(* IEC 61131-3 sources: Building-Automation/Car_Parking_Vending_System/plc, 6 files *)

(* ---- global_vars.st ---- *)
// Global Variables for Car Parking Vending System
// Version: 2.1.0
// Compatible with: Siemens S7-1200/1500, TIA Portal V17+

// =============================================================================
// SYSTEM ENUMERATIONS
// =============================================================================

TYPE SystemState :
(
    INIT := 0,              // System initialization
    IDLE := 1,              // Ready for operation
    PAYMENT := 2,           // Processing payment
    ENTRY := 3,             // Vehicle entry sequence
    PARKING := 4,           // Automated parking
    PARKED := 5,            // Vehicle stored
    RETRIEVAL := 6,         // Vehicle retrieval
    EXIT_SEQUENCE := 7,     // Vehicle exit
    MAINTENANCE := 8,       // Maintenance mode
    EMERGENCY := 9          // Emergency stop
);
END_TYPE;

TYPE ElevatorState :
(
    IDLE := 0,              // Elevator at rest
    MOVING_UP := 1,         // Moving upward
    MOVING_DOWN := 2,       // Moving downward
    POSITIONING := 3,       // Fine positioning
    LOADING := 4,           // Loading vehicle
    UNLOADING := 5,         // Unloading vehicle
    ERROR := 6              // Error state
);
END_TYPE;

TYPE PlatformState :
(
    HOME := 0,              // Home position
    MOVING_X := 1,          // Moving X axis
    MOVING_Y := 2,          // Moving Y axis
    POSITIONING := 3,       // Final positioning
    PICKING_UP := 4,        // Picking up vehicle
    DROPPING_OFF := 5,      // Dropping off vehicle
    ERROR := 6              // Error state
);
END_TYPE;

TYPE PaymentMethod :
(
    NONE := 0,              // No payment
    CASH := 1,              // Cash payment
    CREDIT_CARD := 2,       // Credit/Debit card
    RFID_CARD := 3,         // RFID membership card
    MOBILE_APP := 4,        // Mobile application
    QR_CODE := 5            // QR code payment
);
END_TYPE;

TYPE VehicleSize :
(
    COMPACT := 1,           // Small cars
    STANDARD := 2,          // Standard size
    SUV := 3,               // SUV/Large cars
    MOTORCYCLE := 4         // Motorcycles
);
END_TYPE;

// =============================================================================
// DIGITAL INPUTS (24V DC)
// =============================================================================

VAR_GLOBAL
    // Emergency stops and safety
    I_EmergencyStop_Main        AT %I0.0 : BOOL;   // Main emergency stop
    I_EmergencyStop_Level1      AT %I0.1 : BOOL;   // Level 1 emergency stop
    I_EmergencyStop_Level2      AT %I0.2 : BOOL;   // Level 2 emergency stop
    I_FireDetection_Zone1       AT %I0.3 : BOOL;   // Fire detector zone 1
    I_FireDetection_Zone2       AT %I0.4 : BOOL;   // Fire detector zone 2
    I_FireDetection_Zone3       AT %I0.5 : BOOL;   // Fire detector zone 3

    // Barrier positions
    I_EntryBarrier_OpenLimit    AT %I0.6 : BOOL;   // Entry barrier open
    I_EntryBarrier_CloseLimit   AT %I0.7 : BOOL;   // Entry barrier closed
    I_ExitBarrier_OpenLimit     AT %I1.0 : BOOL;   // Exit barrier open
    I_ExitBarrier_CloseLimit    AT %I1.1 : BOOL;   // Exit barrier closed

    // Vehicle detection
    I_VehiclePresent_Entry      AT %I1.2 : BOOL;   // Vehicle at entry
    I_VehiclePresent_Exit       AT %I1.3 : BOOL;   // Vehicle at exit
    I_VehiclePresent_Platform   AT %I1.4 : BOOL;   // Vehicle on platform
    I_VehiclePresent_Queue      AT %I1.5 : BOOL;   // Vehicle in queue

    // System positions
    I_Elevator1_Home            AT %I1.6 : BOOL;   // Elevator 1 home
    I_Elevator2_Home            AT %I1.7 : BOOL;   // Elevator 2 home
    I_Elevator3_Home            AT %I2.0 : BOOL;   // Elevator 3 home
    I_Platform_Home             AT %I2.1 : BOOL;   // Platform home position

    // System status
    I_DoorInterlocks_AllClosed  AT %I2.2 : BOOL;   // All doors closed
    I_HydraulicSystem_PressureOK AT %I2.3 : BOOL;  // Hydraulic pressure OK
    I_UPS_BatteryOK            AT %I2.4 : BOOL;   // UPS battery status
    I_Ventilation_StatusOK     AT %I2.5 : BOOL;   // Ventilation system OK
    I_MainPower_OK             AT %I2.6 : BOOL;   // Main power status
    I_NetworkConnection_OK     AT %I2.7 : BOOL;   // Network connectivity

    // Payment system inputs
    I_PaymentKiosk_Ready       AT %I3.0 : BOOL;   // Payment kiosk ready
    I_CashInserted             AT %I3.1 : BOOL;   // Cash payment received
    I_CardInserted             AT %I3.2 : BOOL;   // Card inserted
    I_RFIDCardPresent          AT %I3.3 : BOOL;   // RFID card detected
    I_QRCodeScanned            AT %I3.4 : BOOL;   // QR code scanned
    I_TicketPrinter_Ready      AT %I3.5 : BOOL;   // Ticket printer ready
    I_TicketPrinter_PaperOK    AT %I3.6 : BOOL;   // Printer paper OK
    I_ReceiptPrinter_Ready     AT %I3.7 : BOOL;   // Receipt printer ready

END_VAR;

// =============================================================================
// ANALOG INPUTS (4-20mA / 0-10V)
// =============================================================================

VAR_GLOBAL
    // Position feedback
    AI_Elevator1_Position       AT %IW0 : INT;     // Elevator 1 position (mm)
    AI_Elevator2_Position       AT %IW2 : INT;     // Elevator 2 position (mm)
    AI_Elevator3_Position       AT %IW4 : INT;     // Elevator 3 position (mm)
    AI_Platform_XPosition       AT %IW6 : INT;     // Platform X position (mm)
    AI_Platform_YPosition       AT %IW8 : INT;     // Platform Y position (mm)
    AI_Platform_ZPosition       AT %IW10 : INT;    // Platform Z position (mm)

    // System monitoring
    AI_HydraulicPressure        AT %IW12 : INT;    // Hydraulic pressure (bar)
    AI_Temperature_ControlRoom  AT %IW14 : INT;    // Control room temp (°C)
    AI_Humidity_ControlRoom     AT %IW16 : INT;    // Control room humidity (%)
    AI_LoadCell_PlatformWeight  AT %IW18 : INT;    // Platform load (kg)
    AI_PowerConsumption         AT %IW20 : INT;    // Power consumption (kW)
    AI_VibrationLevel          AT %IW22 : INT;    // Vibration level

    // Vehicle dimensions (from laser scanners)
    AI_VehicleLength           AT %IW24 : INT;    // Vehicle length (mm)
    AI_VehicleWidth            AT %IW26 : INT;    // Vehicle width (mm)
    AI_VehicleHeight           AT %IW28 : INT;    // Vehicle height (mm)
    AI_VehicleWeight           AT %IW30 : INT;    // Vehicle weight (kg)

END_VAR;

// =============================================================================
// DIGITAL OUTPUTS (24V DC)
// =============================================================================

VAR_GLOBAL
    // Barrier controls
    Q_EntryBarrier_Open         AT %Q0.0 : BOOL;   // Open entry barrier
    Q_EntryBarrier_Close        AT %Q0.1 : BOOL;   // Close entry barrier
    Q_ExitBarrier_Open          AT %Q0.2 : BOOL;   // Open exit barrier
    Q_ExitBarrier_Close         AT %Q0.3 : BOOL;   // Close exit barrier

    // Elevator controls
    Q_Elevator1_Enable          AT %Q0.4 : BOOL;   // Elevator 1 motor enable
    Q_Elevator2_Enable          AT %Q0.5 : BOOL;   // Elevator 2 motor enable
    Q_Elevator3_Enable          AT %Q0.6 : BOOL;   // Elevator 3 motor enable
    Q_Elevator1_Direction       AT %Q0.7 : BOOL;   // Elevator 1 direction
    Q_Elevator2_Direction       AT %Q1.0 : BOOL;   // Elevator 2 direction
    Q_Elevator3_Direction       AT %Q1.1 : BOOL;   // Elevator 3 direction

    // Platform controls
    Q_Platform_XEnable          AT %Q1.2 : BOOL;   // Platform X axis enable
    Q_Platform_YEnable          AT %Q1.3 : BOOL;   // Platform Y axis enable
    Q_Platform_ZEnable          AT %Q1.4 : BOOL;   // Platform Z axis enable
    Q_Platform_XDirection       AT %Q1.5 : BOOL;   // Platform X direction
    Q_Platform_YDirection       AT %Q1.6 : BOOL;   // Platform Y direction
    Q_Platform_ZDirection       AT %Q1.7 : BOOL;   // Platform Z direction

    // System controls
    Q_HydraulicPump            AT %Q2.0 : BOOL;   // Hydraulic pump start
    Q_VentilationFan           AT %Q2.1 : BOOL;   // Ventilation fan start
    Q_EmergencyLighting        AT %Q2.2 : BOOL;   // Emergency lighting
    Q_MainLighting             AT %Q2.3 : BOOL;   // Main lighting

    // Status indicators
    Q_StatusLight_Green        AT %Q2.4 : BOOL;   // Green status light
    Q_StatusLight_Yellow       AT %Q2.5 : BOOL;   // Yellow status light
    Q_StatusLight_Red          AT %Q2.6 : BOOL;   // Red status light
    Q_AlarmHorn               AT %Q2.7 : BOOL;   // Alarm horn

    // Door locks and safety
    Q_DoorLock_Entry          AT %Q3.0 : BOOL;   // Entry door lock
    Q_DoorLock_Exit           AT %Q3.1 : BOOL;   // Exit door lock
    Q_SafetyReset             AT %Q3.2 : BOOL;   // Safety system reset

    // Payment and printing
    Q_TicketPrinter_Print     AT %Q3.3 : BOOL;   // Print parking ticket
    Q_ReceiptPrinter_Print    AT %Q3.4 : BOOL;   // Print payment receipt
    Q_CashDispenser_Enable    AT %Q3.5 : BOOL;   // Cash change dispenser
    Q_CardReader_Enable       AT %Q3.6 : BOOL;   // Card reader enable
    Q_Display_Enable          AT %Q3.7 : BOOL;   // Customer display enable

    // System status outputs
    Q_SystemReady             AT %Q4.0 : BOOL;   // System ready indicator
    Q_SystemEnabled           AT %Q4.1 : BOOL;   // System enabled
    Q_MaintenanceMode         AT %Q4.2 : BOOL;   // Maintenance mode active
    Q_EmergencyActive         AT %Q4.3 : BOOL;   // Emergency mode active

END_VAR;

// =============================================================================
// ANALOG OUTPUTS (4-20mA / 0-10V)
// =============================================================================

VAR_GLOBAL
    // Speed references
    AQ_Elevator1_SpeedRef       AT %QW0 : INT;     // Elevator 1 speed ref
    AQ_Elevator2_SpeedRef       AT %QW2 : INT;     // Elevator 2 speed ref
    AQ_Elevator3_SpeedRef       AT %QW4 : INT;     // Elevator 3 speed ref
    AQ_Platform_XSpeedRef       AT %QW6 : INT;     // Platform X speed ref
    AQ_Platform_YSpeedRef       AT %QW8 : INT;     // Platform Y speed ref
    AQ_Platform_ZSpeedRef       AT %QW10 : INT;    // Platform Z speed ref

    // System controls
    AQ_HydraulicPressureRef     AT %QW12 : INT;    // Hydraulic pressure ref
    AQ_VentilationSpeedRef      AT %QW14 : INT;    // Ventilation speed ref
    AQ_LightingLevel           AT %QW16 : INT;    // Lighting level control

END_VAR;

// =============================================================================
// DATA STRUCTURES
// =============================================================================

TYPE ParkingSpace :
STRUCT
    Level : INT;                // Parking level (1-15)
    Position : INT;             // Position on level (1-20)
    Occupied : BOOL;            // Space occupied flag
    VehicleID : STRING[20];     // Vehicle identification
    ParkingTime : DATE_AND_TIME; // Time when parked
    VehicleType : VehicleSize;   // Vehicle size category
    ReservedFor : STRING[50];    // Reserved for specific customer
    MaintenanceRequired : BOOL;  // Maintenance flag
END_STRUCT;
END_TYPE;

TYPE Transaction :
STRUCT
    TransactionID : DINT;       // Unique transaction ID
    Timestamp : DATE_AND_TIME;  // Transaction timestamp
    CustomerID : STRING[50];    // Customer identification
    VehicleID : STRING[20];     // Vehicle license plate
    PaymentMethod : PaymentMethod; // Payment type used
    Amount : REAL;              // Payment amount
    ParkingDuration : TIME;     // Requested parking duration
    SpaceAssigned : ParkingSpace; // Assigned parking space
    Status : STRING[20];        // Transaction status
END_STRUCT;
END_TYPE;

TYPE SystemStatistics :
STRUCT
    TotalVehiclesParked : DINT;     // Total vehicles parked
    TotalVehiclesRetrieved : DINT;  // Total vehicles retrieved
    TotalRevenue : REAL;            // Total revenue generated
    AverageParkingTime : TIME;      // Average parking operation time
    AverageRetrievalTime : TIME;    // Average retrieval operation time
    SystemUptime : TIME;            // Total system uptime
    MaintenanceHours : TIME;        // Total maintenance time
    EmergencyStops : INT;           // Number of emergency stops
    PowerFailures : INT;            // Number of power failures
    LastMaintenanceDate : DATE;     // Last maintenance date
END_STRUCT;
END_TYPE;

TYPE ElevatorData :
STRUCT
    CurrentLevel : INT;         // Current elevator level
    TargetLevel : INT;          // Target level
    CurrentPosition : REAL;     // Current position (mm)
    TargetPosition : REAL;      // Target position (mm)
    Speed : REAL;               // Current speed (mm/s)
    State : ElevatorState;      // Current state
    LoadWeight : REAL;          // Current load weight (kg)
    LastService : DATE;         // Last service date
    OperationHours : TIME;      // Total operation hours
    FaultCode : INT;            // Current fault code
    Available : BOOL;           // Elevator available
END_STRUCT;
END_TYPE;

TYPE PlatformData :
STRUCT
    XPosition : REAL;           // Current X position (mm)
    YPosition : REAL;           // Current Y position (mm)
    ZPosition : REAL;           // Current Z position (mm)
    XTarget : REAL;             // Target X position
    YTarget : REAL;             // Target Y position
    ZTarget : REAL;             // Target Z position
    State : PlatformState;      // Current platform state
    LoadWeight : REAL;          // Current load weight (kg)
    VehicleSecured : BOOL;      // Vehicle properly secured
    LastCalibration : DATE_AND_TIME; // Last calibration
    FaultCode : INT;            // Current fault code
    Available : BOOL;           // Platform available
END_STRUCT;
END_TYPE;

// =============================================================================
// GLOBAL SYSTEM VARIABLES
// =============================================================================

VAR_GLOBAL
    // Parking space array (15 levels × 20 spaces = 300 total)
    ParkingSpaces : ARRAY[1..15, 1..20] OF ParkingSpace;

    // System statistics and monitoring
    SystemStats : SystemStatistics;

    // Equipment data
    Elevator1 : ElevatorData;
    Elevator2 : ElevatorData;
    Elevator3 : ElevatorData;
    Platform : PlatformData;

    // Current transaction
    CurrentTransaction : Transaction;
    TransactionCounter : DINT := 0;

    // System configuration
    MaxVehicleLength : REAL := 5200.0;     // mm
    MaxVehicleWidth : REAL := 2100.0;      // mm
    MaxVehicleHeight : REAL := 1800.0;     // mm
    MaxVehicleWeight : REAL := 3500.0;     // kg

    // Pricing structure
    HourlyRate : REAL := 2.50;             // Currency per hour
    DailyRate : REAL := 15.00;             // Currency per day
    MonthlyRate : REAL := 150.00;          // Currency per month

    // Operating parameters
    ElevatorSpeed : REAL := 2500.0;        // mm/s
    PlatformSpeed : REAL := 1500.0;        // mm/s
    PositioningTolerance : REAL := 5.0;    // mm

    // System timers and counters
    SystemStartTime : DATE_AND_TIME;
    LastTransactionTime : DATE_AND_TIME;
    NextMaintenanceTime : DATE_AND_TIME;

    // Queue management
    WaitingVehicles : INT := 0;
    MaxQueueLength : INT := 10;
    EstimatedWaitTime : TIME;

    // Performance monitoring
    SystemEfficiency : REAL;               // 0-100%
    EnergyConsumption : REAL;              // kWh
    ThroughputPerHour : REAL;              // vehicles/hour

    // Alarm and event logging
    AlarmBuffer : ARRAY[1..100] OF STRING[200];
    EventBuffer : ARRAY[1..1000] OF STRING[200];
    AlarmIndex : INT := 0;
    EventIndex : INT := 0;

    // Communication and networking
    HMI_Connected : BOOL := FALSE;
    Database_Connected : BOOL := FALSE;
    PaymentGateway_Connected : BOOL := FALSE;
    RemoteMonitoring_Connected : BOOL := FALSE;

    // Weather and environmental
    OutdoorTemperature : REAL;
    WindSpeed : REAL;
    RainIntensity : REAL;

END_VAR;

// =============================================================================
// SYSTEM CONSTANTS
// =============================================================================

VAR_GLOBAL CONSTANT
    SYSTEM_VERSION : STRING := '2.1.0';
    MAX_PARKING_LEVELS : INT := 15;
    SPACES_PER_LEVEL : INT := 20;
    TOTAL_PARKING_SPACES : INT := 300;

    // Safety limits
    MAX_ELEVATOR_SPEED : REAL := 3000.0;   // mm/s
    MAX_PLATFORM_SPEED : REAL := 2000.0;   // mm/s
    EMERGENCY_STOP_TIME : TIME := T#2s;

    // Operational timeouts
    PAYMENT_TIMEOUT : TIME := T#120s;
    ENTRY_TIMEOUT : TIME := T#60s;
    PARKING_TIMEOUT : TIME := T#300s;
    RETRIEVAL_TIMEOUT : TIME := T#300s;
    EXIT_TIMEOUT : TIME := T#90s;

    // Communication timeouts
    HMI_TIMEOUT : TIME := T#10s;
    DATABASE_TIMEOUT : TIME := T#30s;
    NETWORK_TIMEOUT : TIME := T#15s;

END_VAR;

(* ---- elevator_controller.st ---- *)
FUNCTION_BLOCK ElevatorController
VAR_INPUT
    ElevatorNumber : INT;               // Elevator number (1, 2, or 3)
    TargetLevel : INT;                  // Target level (1-15)
    Execute : BOOL;                     // Execute movement command
    Stop : BOOL;                        // Emergency stop
    Reset : BOOL;                       // Reset elevator
    ManualMode : BOOL;                  // Manual operation mode
    ManualDirection : BOOL;             // Manual direction (TRUE=up, FALSE=down)
    ManualSpeed : REAL;                 // Manual speed reference
END_VAR

VAR_OUTPUT
    Done : BOOL;                        // Movement completed
    Busy : BOOL;                        // Movement in progress
    Error : BOOL;                       // Error condition
    ErrorID : INT;                      // Error identification code
    CurrentLevel : INT;                 // Current elevator level
    CurrentPosition : REAL;             // Current position (mm)
    AtLevel : BOOL;                     // At target level
    DoorOpen : BOOL;                    // Door open status
    Available : BOOL;                   // Elevator available for use
    LoadWeight : REAL;                  // Current load weight
    MotorSpeed : REAL;                  // Current motor speed
END_VAR

VAR
    // Control state machine
    state : INT := 0;
    previousState : INT;
    stateTimer : TON;
    movementTimer : TON;

    // Position and motion control
    currentPos : REAL;                  // Current position in mm
    targetPos : REAL;                   // Target position in mm
    homePosition : REAL := 0.0;         // Ground level position
    levelHeight : REAL := 3000.0;       // Height per level (mm)
    positionTolerance : REAL := 20.0;   // Position tolerance (mm)

    // Motion parameters
    maxSpeed : REAL := 2500.0;          // Maximum speed (mm/s)
    acceleration : REAL := 500.0;       // Acceleration (mm/s²)
    deceleration : REAL := 750.0;       // Deceleration (mm/s²)
    currentSpeed : REAL := 0.0;         // Current speed
    targetSpeed : REAL := 0.0;          // Target speed

    // Safety and monitoring
    safetyOK : BOOL := TRUE;
    overloadDetected : BOOL := FALSE;
    doorInterlockOK : BOOL := TRUE;
    emergencyStopActive : BOOL := FALSE;

    // Door control
    doorState : INT := 0;               // 0=closed, 1=opening, 2=open, 3=closing
    doorTimer : TON;
    doorTimeout : TIME := T#10s;

    // Maintenance and diagnostics
    totalOperationTime : TIME;
    totalDistance : REAL := 0.0;
    cycleCount : DINT := 0;
    lastMaintenanceDistance : REAL := 0.0;
    maintenanceRequired : BOOL := FALSE;

    // Error handling
    errorHistory : ARRAY[1..10] OF INT;
    errorIndex : INT := 1;
    retryCount : INT := 0;
    maxRetries : INT := 3;

    // Performance monitoring
    averageSpeed : REAL;
    lastMovementTime : TIME;
    efficiency : REAL := 100.0;

END_VAR

// Input validation
IF ElevatorNumber < 1 OR ElevatorNumber > 3 THEN
    Error := TRUE;
    ErrorID := 5001; // Invalid elevator number
    Available := FALSE;
    RETURN;
END_IF;

IF TargetLevel < 1 OR TargetLevel > MAX_PARKING_LEVELS THEN
    Error := TRUE;
    ErrorID := 5002; // Invalid target level
    RETURN;
END_IF;

// Get current position based on elevator number
CASE ElevatorNumber OF
    1: currentPos := SCALE_INT_TO_REAL(AI_Elevator1_Position, 0.0, 45000.0);
    2: currentPos := SCALE_INT_TO_REAL(AI_Elevator2_Position, 0.0, 45000.0);
    3: currentPos := SCALE_INT_TO_REAL(AI_Elevator3_Position, 0.0, 45000.0);
END_CASE;

CurrentPosition := currentPos;
LoadWeight := SCALE_INT_TO_REAL(AI_LoadCell_PlatformWeight, 0.0, 5000.0);

// Calculate current level
CurrentLevel := REAL_TO_INT((currentPos / levelHeight) + 1);
IF CurrentLevel < 1 THEN CurrentLevel := 1; END_IF;
IF CurrentLevel > MAX_PARKING_LEVELS THEN CurrentLevel := MAX_PARKING_LEVELS; END_IF;

// Safety checks
safetyOK := NOT I_EmergencyStop_Main AND
            NOT I_EmergencyStop_Level1 AND
            NOT I_EmergencyStop_Level2 AND
            I_HydraulicSystem_PressureOK AND
            I_UPS_BatteryOK;

overloadDetected := LoadWeight > 4000.0; // 4000kg limit
doorInterlockOK := I_DoorInterlocks_AllClosed;
emergencyStopActive := Stop OR NOT safetyOK;

// Emergency stop handling
IF emergencyStopActive THEN
    state := 90; // Emergency stop state
    targetSpeed := 0.0;
    Error := TRUE;
    ErrorID := 5010;
END_IF;

// Reset handling
IF Reset AND state = 90 THEN
    state := 0; // Reset to idle
    Error := FALSE;
    ErrorID := 0;
    retryCount := 0;
END_IF;

// Calculate target position
targetPos := (TargetLevel - 1) * levelHeight;

// Check if at target level
AtLevel := ABS(currentPos - targetPos) <= positionTolerance;

// Execute movement command
IF Execute AND NOT Busy AND state = 0 AND safetyOK THEN
    IF NOT AtLevel THEN
        Busy := TRUE;
        Done := FALSE;
        state := 10; // Start movement
        movementTimer(IN := TRUE, PT := T#0s);
        cycleCount := cycleCount + 1;
    ELSE
        Done := TRUE; // Already at target
    END_IF;
END_IF;

// Manual mode handling
IF ManualMode AND state = 0 AND safetyOK THEN
    state := 80; // Manual mode
    Busy := TRUE;
END_IF;

// Main state machine
CASE state OF

    0: // IDLE
        Busy := FALSE;
        Available := TRUE AND safetyOK AND NOT maintenanceRequired;
        targetSpeed := 0.0;

        // Check for maintenance requirements
        IF (totalDistance - lastMaintenanceDistance) > 100000000.0 THEN // 100km
            maintenanceRequired := TRUE;
            Available := FALSE;
        END_IF;

    // =============================================================================
    // MOVEMENT SEQUENCE (States 10-49)
    // =============================================================================

    10: // PREPARE_FOR_MOVEMENT
        Available := FALSE;

        // Ensure doors are closed
        IF NOT doorInterlockOK THEN
            state := 11; // Close doors first
        ELSE
            state := 12; // Doors already closed
        END_IF;

    11: // CLOSE_DOORS
        doorState := 3; // Closing
        doorTimer(IN := TRUE, PT := doorTimeout);

        IF doorInterlockOK THEN
            doorState := 0; // Closed
            state := 12;
            doorTimer(IN := FALSE);
        ELSIF doorTimer.Q THEN
            Error := TRUE;
            ErrorID := 5011; // Door close timeout
            state := 91;
            doorTimer(IN := FALSE);
        END_IF;

    12: // START_MOVEMENT
        // Enable motor based on elevator number
        CASE ElevatorNumber OF
            1: Q_Elevator1_Enable := TRUE;
            2: Q_Elevator2_Enable := TRUE;
            3: Q_Elevator3_Enable := TRUE;
        END_CASE;

        // Determine direction
        IF targetPos > currentPos THEN
            // Moving up
            CASE ElevatorNumber OF
                1: Q_Elevator1_Direction := TRUE;
                2: Q_Elevator2_Direction := TRUE;
                3: Q_Elevator3_Direction := TRUE;
            END_CASE;
        ELSE
            // Moving down
            CASE ElevatorNumber OF
                1: Q_Elevator1_Direction := FALSE;
                2: Q_Elevator2_Direction := FALSE;
                3: Q_Elevator3_Direction := FALSE;
            END_CASE;
        END_IF;

        state := 13; // Accelerate

    13: // ACCELERATE
        // Calculate required speed
        IF ABS(targetPos - currentPos) > 1000.0 THEN
            targetSpeed := maxSpeed; // Full speed for long distances
        ELSE
            targetSpeed := maxSpeed * 0.5; // Half speed for short distances
        END_IF;

        // Accelerate to target speed
        IF currentSpeed < targetSpeed THEN
            currentSpeed := currentSpeed + (acceleration * 0.1); // 100ms cycle
            IF currentSpeed > targetSpeed THEN
                currentSpeed := targetSpeed;
            END_IF;
        END_IF;

        // Check if close to target for deceleration
        IF ABS(targetPos - currentPos) <= (currentSpeed * currentSpeed) / (2.0 * deceleration) THEN
            state := 14; // Start deceleration
        END_IF;

        // Safety check during movement
        IF NOT safetyOK OR overloadDetected THEN
            state := 90; // Emergency stop
        END_IF;

    14: // DECELERATE
        // Calculate deceleration distance
        targetSpeed := SQRT(2.0 * deceleration * ABS(targetPos - currentPos));

        IF targetSpeed < 100.0 THEN
            targetSpeed := 100.0; // Minimum speed for positioning
        END_IF;

        // Decelerate
        IF currentSpeed > targetSpeed THEN
            currentSpeed := currentSpeed - (deceleration * 0.1);
            IF currentSpeed < targetSpeed THEN
                currentSpeed := targetSpeed;
            END_IF;
        END_IF;

        // Check if at target position
        IF ABS(targetPos - currentPos) <= positionTolerance THEN
            state := 15; // Stop
        END_IF;

        // Timeout check
        IF movementTimer.ET > T#300s THEN
            Error := TRUE;
            ErrorID := 5012; // Movement timeout
            state := 91;
        END_IF;

    15: // STOP_AT_TARGET
        targetSpeed := 0.0;
        currentSpeed := 0.0;

        // Stop motor
        CASE ElevatorNumber OF
            1: Q_Elevator1_Enable := FALSE;
            2: Q_Elevator2_Enable := FALSE;
            3: Q_Elevator3_Enable := FALSE;
        END_CASE;

        stateTimer(IN := TRUE, PT := T#2s);

        IF stateTimer.Q THEN
            state := 16; // Final positioning
            stateTimer(IN := FALSE);
        END_IF;

    16: // FINE_POSITIONING
        // Fine positioning at very low speed
        IF ABS(targetPos - currentPos) > 5.0 THEN
            CASE ElevatorNumber OF
                1: Q_Elevator1_Enable := TRUE;
                2: Q_Elevator2_Enable := TRUE;
                3: Q_Elevator3_Enable := TRUE;
            END_CASE;

            currentSpeed := 50.0; // Very slow speed
            targetSpeed := 50.0;
        ELSE
            state := 17; // Positioning complete
        END_IF;

        stateTimer(IN := TRUE, PT := T#30s);
        IF stateTimer.Q THEN
            state := 17; // Timeout - accept current position
            stateTimer(IN := FALSE);
        END_IF;

    17: // POSITIONING_COMPLETE
        // Final stop
        targetSpeed := 0.0;
        currentSpeed := 0.0;

        CASE ElevatorNumber OF
            1: Q_Elevator1_Enable := FALSE;
            2: Q_Elevator2_Enable := FALSE;
            3: Q_Elevator3_Enable := FALSE;
        END_CASE;

        // Update statistics
        lastMovementTime := movementTimer.ET;
        totalDistance := totalDistance + ABS(targetPos - currentPos);
        averageSpeed := ABS(targetPos - currentPos) / TIME_TO_REAL(lastMovementTime);

        state := 20; // Open doors

    20: // OPEN_DOORS
        doorState := 1; // Opening
        doorTimer(IN := TRUE, PT := doorTimeout);

        stateTimer(IN := TRUE, PT := T#2s);

        IF stateTimer.Q THEN
            doorState := 2; // Open
            DoorOpen := TRUE;
            state := 30; // Movement complete
            doorTimer(IN := FALSE);
            stateTimer(IN := FALSE);
        ELSIF doorTimer.Q THEN
            // Door open timeout - continue anyway
            DoorOpen := FALSE;
            state := 30;
            doorTimer(IN := FALSE);
        END_IF;

    30: // MOVEMENT_COMPLETE
        Done := TRUE;
        Busy := FALSE;
        Available := TRUE;
        AtLevel := TRUE;

        // Log successful movement
        LogEvent('ELEVATOR_MOVEMENT', 'Elevator ' + INT_TO_STRING(ElevatorNumber) +
                 ' moved to level ' + INT_TO_STRING(TargetLevel) +
                 ' in ' + TIME_TO_STRING(lastMovementTime));

        state := 0; // Return to idle

    // =============================================================================
    // MANUAL MODE (States 80-89)
    // =============================================================================

    80: // MANUAL_OPERATION
        Available := FALSE;

        IF NOT ManualMode THEN
            state := 0; // Exit manual mode
            targetSpeed := 0.0;
        ELSE
            // Enable motor
            CASE ElevatorNumber OF
                1: Q_Elevator1_Enable := TRUE;
                   Q_Elevator1_Direction := ManualDirection;
                2: Q_Elevator2_Enable := TRUE;
                   Q_Elevator2_Direction := ManualDirection;
                3: Q_Elevator3_Enable := TRUE;
                   Q_Elevator3_Direction := ManualDirection;
            END_CASE;

            targetSpeed := ManualSpeed;
            currentSpeed := ManualSpeed;

            // Safety limits in manual mode
            IF currentPos <= 0.0 AND NOT ManualDirection THEN
                targetSpeed := 0.0; // At bottom limit
            ELSIF currentPos >= 45000.0 AND ManualDirection THEN
                targetSpeed := 0.0; // At top limit
            END_IF;
        END_IF;

    // =============================================================================
    // ERROR STATES (States 90-99)
    // =============================================================================

    90: // EMERGENCY_STOP
        targetSpeed := 0.0;
        currentSpeed := 0.0;
        Available := FALSE;
        Error := TRUE;

        // Stop motor immediately
        CASE ElevatorNumber OF
            1: Q_Elevator1_Enable := FALSE;
            2: Q_Elevator2_Enable := FALSE;
            3: Q_Elevator3_Enable := FALSE;
        END_CASE;

        // Log emergency stop
        LogError(ErrorID, 'Emergency stop - Elevator ' + INT_TO_STRING(ElevatorNumber));

        // Stay in this state until reset

    91: // ERROR_WITH_RETRY
        Error := TRUE;
        Available := FALSE;
        targetSpeed := 0.0;

        // Stop motor
        CASE ElevatorNumber OF
            1: Q_Elevator1_Enable := FALSE;
            2: Q_Elevator2_Enable := FALSE;
            3: Q_Elevator3_Enable := FALSE;
        END_CASE;

        // Record error
        errorHistory[errorIndex] := ErrorID;
        errorIndex := errorIndex + 1;
        IF errorIndex > 10 THEN errorIndex := 1; END_IF;

        // Retry logic
        IF retryCount < maxRetries AND safetyOK THEN
            retryCount := retryCount + 1;
            stateTimer(IN := TRUE, PT := T#10s);

            IF stateTimer.Q THEN
                state := 10; // Retry movement
                Error := FALSE;
                ErrorID := 0;
                stateTimer(IN := FALSE);
            END_IF;
        ELSE
            state := 90; // Give up, require manual reset
        END_IF;

END_CASE;

// Set speed reference outputs
CASE ElevatorNumber OF
    1: AQ_Elevator1_SpeedRef := REAL_TO_INT(currentSpeed);
    2: AQ_Elevator2_SpeedRef := REAL_TO_INT(currentSpeed);
    3: AQ_Elevator3_SpeedRef := REAL_TO_INT(currentSpeed);
END_CASE;

// Update motor speed output for monitoring
MotorSpeed := currentSpeed;

// Update total operation time
totalOperationTime := totalOperationTime + T#100ms;

// Update elevator data structure
CASE ElevatorNumber OF
    1: Elevator1.CurrentLevel := CurrentLevel;
       Elevator1.CurrentPosition := currentPos;
       Elevator1.TargetLevel := TargetLevel;
       Elevator1.TargetPosition := targetPos;
       Elevator1.Speed := currentSpeed;
       Elevator1.LoadWeight := LoadWeight;
       Elevator1.Available := Available;
       Elevator1.FaultCode := ErrorID;
       Elevator1.OperationHours := totalOperationTime;

    2: Elevator2.CurrentLevel := CurrentLevel;
       Elevator2.CurrentPosition := currentPos;
       Elevator2.TargetLevel := TargetLevel;
       Elevator2.TargetPosition := targetPos;
       Elevator2.Speed := currentSpeed;
       Elevator2.LoadWeight := LoadWeight;
       Elevator2.Available := Available;
       Elevator2.FaultCode := ErrorID;
       Elevator2.OperationHours := totalOperationTime;

    3: Elevator3.CurrentLevel := CurrentLevel;
       Elevator3.CurrentPosition := currentPos;
       Elevator3.TargetLevel := TargetLevel;
       Elevator3.TargetPosition := targetPos;
       Elevator3.Speed := currentSpeed;
       Elevator3.LoadWeight := LoadWeight;
       Elevator3.Available := Available;
       Elevator3.FaultCode := ErrorID;
       Elevator3.OperationHours := totalOperationTime;
END_CASE;

// Store previous state for debugging
previousState := state;

END_FUNCTION_BLOCK

(* ---- parking_controller.st ---- *)
FUNCTION_BLOCK ParkingController
VAR_INPUT
    Execute : BOOL;                     // Execute parking sequence
    VehicleRetrievalRequest : BOOL;     // Vehicle retrieval request
    CustomerID : STRING[50];            // Customer identification
    VehicleID : STRING[20];             // Vehicle license plate
    PaymentValidated : BOOL;            // Payment validation status
END_VAR

VAR_OUTPUT
    Done : BOOL;                        // Operation completed
    Busy : BOOL;                        // Operation in progress
    Error : BOOL;                       // Error occurred
    ErrorID : INT;                      // Error identification
    AssignedSpace : ParkingSpace;       // Assigned parking space
    EstimatedTime : TIME;               // Estimated completion time
END_VAR

VAR
    // State machine for parking operations
    state : INT := 0;
    stepTimer : TON;
    operationTimer : TON;

    // Vehicle handling
    vehicleDimensions : VehicleDimensions;
    optimalSpace : ParkingSpace;
    selectedElevator : INT;

    // Position control
    targetLevel : INT;
    targetXPosition : REAL;
    targetYPosition : REAL;
    currentOperation : STRING[50];

    // Safety and monitoring
    platformSecure : BOOL;
    elevatorReady : BOOL;
    spaceAvailable : BOOL;

    // Performance tracking
    operationStartTime : DATE_AND_TIME;
    parkingSequenceTime : TIME;
    retrievalSequenceTime : TIME;

    // Error handling
    retryCount : INT := 0;
    maxRetries : INT := 3;
    lastErrorTime : DATE_AND_TIME;

END_VAR

// Vehicle dimensions structure
TYPE VehicleDimensions :
STRUCT
    Length : REAL;
    Width : REAL;
    Height : REAL;
    Weight : REAL;
    VehicleType : VehicleSize;
END_STRUCT;
END_TYPE;

// Main execution logic
IF Execute AND NOT Busy THEN
    Busy := TRUE;
    Done := FALSE;
    Error := FALSE;
    state := 10; // Start parking sequence
    operationStartTime := GetSystemTime();
    operationTimer(IN := TRUE, PT := T#0s);
ELSIF VehicleRetrievalRequest AND NOT Busy THEN
    Busy := TRUE;
    Done := FALSE;
    Error := FALSE;
    state := 50; // Start retrieval sequence
    operationStartTime := GetSystemTime();
    operationTimer(IN := TRUE, PT := T#0s);
END_IF;

// Main state machine
CASE state OF

    0: // IDLE
        Busy := FALSE;
        Done := FALSE;
        Error := FALSE;
        currentOperation := 'IDLE';

    // =============================================================================
    // PARKING SEQUENCE (States 10-39)
    // =============================================================================

    10: // SCAN_VEHICLE_DIMENSIONS
        currentOperation := 'SCANNING_VEHICLE';

        // Get vehicle dimensions from laser scanners
        vehicleDimensions.Length := SCALE_INT_TO_REAL(AI_VehicleLength, 0.0, 6000.0);
        vehicleDimensions.Width := SCALE_INT_TO_REAL(AI_VehicleWidth, 0.0, 2500.0);
        vehicleDimensions.Height := SCALE_INT_TO_REAL(AI_VehicleHeight, 0.0, 2000.0);
        vehicleDimensions.Weight := SCALE_INT_TO_REAL(AI_VehicleWeight, 0.0, 5000.0);

        // Determine vehicle type
        IF vehicleDimensions.Length <= 4200.0 AND vehicleDimensions.Width <= 1800.0 THEN
            vehicleDimensions.VehicleType := COMPACT;
        ELSIF vehicleDimensions.Length <= 5200.0 AND vehicleDimensions.Width <= 2100.0 THEN
            vehicleDimensions.VehicleType := STANDARD;
        ELSIF vehicleDimensions.Height <= 1200.0 THEN
            vehicleDimensions.VehicleType := MOTORCYCLE;
        ELSE
            vehicleDimensions.VehicleType := SUV;
        END_IF;

        // Validate vehicle dimensions
        IF vehicleDimensions.Length > MaxVehicleLength OR
           vehicleDimensions.Width > MaxVehicleWidth OR
           vehicleDimensions.Height > MaxVehicleHeight OR
           vehicleDimensions.Weight > MaxVehicleWeight THEN
            Error := TRUE;
            ErrorID := 2001; // Vehicle too large
            state := 90; // Error handling
        ELSE
            state := 11; // Continue to space finding
        END_IF;

    11: // FIND_OPTIMAL_SPACE
        currentOperation := 'FINDING_PARKING_SPACE';

        IF FindOptimalParkingSpace() THEN
            state := 12; // Space found
        ELSE
            Error := TRUE;
            ErrorID := 2002; // No available space
            state := 90; // Error handling
        END_IF;

    12: // PREPARE_PLATFORM
        currentOperation := 'PREPARING_PLATFORM';

        // Ensure platform is at home position
        IF I_Platform_Home THEN
            Q_Platform_XEnable := TRUE;
            Q_Platform_YEnable := TRUE;
            Q_Platform_ZEnable := TRUE;
            state := 13;
        ELSE
            // Move platform to home position
            MovePlatformToHome();
        END_IF;

    13: // POSITION_VEHICLE_ON_PLATFORM
        currentOperation := 'POSITIONING_VEHICLE';

        stepTimer(IN := TRUE, PT := T#30s);

        // Check if vehicle is properly positioned
        IF I_VehiclePresent_Platform AND
           ABS(AI_Platform_XPosition - 3000) < 50 AND  // Center X position
           ABS(AI_Platform_YPosition - 7500) < 50 THEN // Center Y position
            platformSecure := TRUE;
            state := 14;
            stepTimer(IN := FALSE);
        ELSIF stepTimer.Q THEN
            Error := TRUE;
            ErrorID := 2003; // Vehicle positioning timeout
            state := 90;
            stepTimer(IN := FALSE);
        END_IF;

    14: // SECURE_VEHICLE
        currentOperation := 'SECURING_VEHICLE';

        // Activate platform securing mechanisms
        Q_Platform_ZEnable := TRUE;
        AQ_Platform_ZSpeedRef := 100; // Slow speed for securing

        stepTimer(IN := TRUE, PT := T#10s);

        // Check if vehicle is secured (weight on platform)
        IF AI_LoadCell_PlatformWeight > 500 THEN // Minimum 500kg
            Platform.VehicleSecured := TRUE;
            state := 15;
            stepTimer(IN := FALSE);
        ELSIF stepTimer.Q THEN
            Error := TRUE;
            ErrorID := 2004; // Vehicle securing failed
            state := 90;
            stepTimer(IN := FALSE);
        END_IF;

    15: // SELECT_ELEVATOR
        currentOperation := 'SELECTING_ELEVATOR';

        selectedElevator := SelectOptimalElevator();

        IF selectedElevator > 0 THEN
            state := 16;
        ELSE
            Error := TRUE;
            ErrorID := 2005; // No elevator available
            state := 90;
        END_IF;

    16: // MOVE_TO_ELEVATOR
        currentOperation := 'MOVING_TO_ELEVATOR';

        // Calculate elevator loading position
        CASE selectedElevator OF
            1: targetXPosition := 1500.0; // Elevator 1 position
            2: targetXPosition := 3000.0; // Elevator 2 position
            3: targetXPosition := 4500.0; // Elevator 3 position
        END_CASE;

        targetYPosition := 2000.0; // Elevator loading position

        MovePlatformToPosition(targetXPosition, targetYPosition, 0.0);

        // Check if platform reached elevator
        IF ABS(AI_Platform_XPosition - targetXPosition) < 20 AND
           ABS(AI_Platform_YPosition - targetYPosition) < 20 THEN
            state := 17;
        END_IF;

    17: // LOAD_INTO_ELEVATOR
        currentOperation := 'LOADING_INTO_ELEVATOR';

        stepTimer(IN := TRUE, PT := T#60s);

        // Enable selected elevator
        CASE selectedElevator OF
            1: Q_Elevator1_Enable := TRUE;
            2: Q_Elevator2_Enable := TRUE;
            3: Q_Elevator3_Enable := TRUE;
        END_CASE;

        // Transfer vehicle to elevator
        Q_Platform_YEnable := TRUE;
        Q_Platform_YDirection := TRUE; // Move forward into elevator
        AQ_Platform_YSpeedRef := 500; // Slow speed for precision

        // Check if loading complete
        IF ABS(AI_Platform_YPosition - 1000.0) < 10 THEN // Inside elevator
            state := 18;
            stepTimer(IN := FALSE);
        ELSIF stepTimer.Q THEN
            Error := TRUE;
            ErrorID := 2006; // Elevator loading timeout
            state := 90;
            stepTimer(IN := FALSE);
        END_IF;

    18: // MOVE_TO_PARKING_LEVEL
        currentOperation := 'MOVING_TO_LEVEL';

        targetLevel := optimalSpace.Level;

        MoveElevatorToLevel(selectedElevator, targetLevel);

        // Check if elevator reached target level
        CASE selectedElevator OF
            1: IF ABS(AI_Elevator1_Position - (targetLevel * 3000)) < 50 THEN
                   state := 19;
               END_IF;
            2: IF ABS(AI_Elevator2_Position - (targetLevel * 3000)) < 50 THEN
                   state := 19;
               END_IF;
            3: IF ABS(AI_Elevator3_Position - (targetLevel * 3000)) < 50 THEN
                   state := 19;
               END_IF;
        END_CASE;

    19: // UNLOAD_FROM_ELEVATOR
        currentOperation := 'UNLOADING_FROM_ELEVATOR';

        stepTimer(IN := TRUE, PT := T#60s);

        // Move platform out of elevator to parking level
        Q_Platform_YDirection := FALSE; // Move backward out of elevator
        AQ_Platform_YSpeedRef := 500; // Slow speed

        // Calculate target position on parking level
        targetXPosition := optimalSpace.Position * 300.0; // 300mm spacing
        targetYPosition := 7500.0; // Level corridor position

        IF ABS(AI_Platform_YPosition - targetYPosition) < 20 THEN
            state := 20;
            stepTimer(IN := FALSE);
        ELSIF stepTimer.Q THEN
            Error := TRUE;
            ErrorID := 2007; // Elevator unloading timeout
            state := 90;
            stepTimer(IN := FALSE);
        END_IF;

    20: // MOVE_TO_PARKING_SPACE
        currentOperation := 'MOVING_TO_SPACE';

        MovePlatformToPosition(targetXPosition, targetYPosition, 0.0);

        // Check if platform reached parking space
        IF ABS(AI_Platform_XPosition - targetXPosition) < 10 AND
           ABS(AI_Platform_YPosition - targetYPosition) < 10 THEN
            state := 21;
        END_IF;

    21: // DEPOSIT_VEHICLE
        currentOperation := 'DEPOSITING_VEHICLE';

        stepTimer(IN := TRUE, PT := T#30s);

        // Lower platform to deposit vehicle
        Q_Platform_ZDirection := FALSE; // Move down
        AQ_Platform_ZSpeedRef := 200; // Very slow for safety

        // Check if vehicle deposited (reduced weight on platform)
        IF AI_LoadCell_PlatformWeight < 100 THEN // Most weight removed
            state := 22;
            stepTimer(IN := FALSE);
        ELSIF stepTimer.Q THEN
            Error := TRUE;
            ErrorID := 2008; // Vehicle deposit timeout
            state := 90;
            stepTimer(IN := FALSE);
        END_IF;

    22: // UPDATE_PARKING_RECORD
        currentOperation := 'UPDATING_RECORDS';

        // Mark space as occupied
        ParkingSpaces[optimalSpace.Level, optimalSpace.Position].Occupied := TRUE;
        ParkingSpaces[optimalSpace.Level, optimalSpace.Position].VehicleID := VehicleID;
        ParkingSpaces[optimalSpace.Level, optimalSpace.Position].ParkingTime := GetSystemTime();
        ParkingSpaces[optimalSpace.Level, optimalSpace.Position].VehicleType := vehicleDimensions.VehicleType;

        // Update transaction record
        CurrentTransaction.SpaceAssigned := optimalSpace;
        CurrentTransaction.Status := 'PARKED';

        // Update system statistics
        SystemStats.TotalVehiclesParked := SystemStats.TotalVehiclesParked + 1;
        parkingSequenceTime := operationTimer.ET;

        // Calculate average parking time
        SystemStats.AverageParkingTime :=
            DINT_TO_TIME((TIME_TO_DINT(SystemStats.AverageParkingTime) *
                         (SystemStats.TotalVehiclesParked - 1) +
                         TIME_TO_DINT(parkingSequenceTime)) /
                         SystemStats.TotalVehiclesParked);

        state := 23; // Return platform home

    23: // RETURN_PLATFORM_HOME
        currentOperation := 'RETURNING_HOME';

        MovePlatformToHome();

        IF I_Platform_Home THEN
            state := 30; // Parking sequence complete
        END_IF;

    30: // PARKING_COMPLETE
        currentOperation := 'PARKING_COMPLETE';
        AssignedSpace := optimalSpace;
        Done := TRUE;
        Busy := FALSE;
        state := 0; // Return to idle

        // Log successful parking
        LogEvent('PARKING_SUCCESS', VehicleID + ' parked at Level ' +
                 INT_TO_STRING(optimalSpace.Level) + ' Position ' +
                 INT_TO_STRING(optimalSpace.Position));

    // =============================================================================
    // RETRIEVAL SEQUENCE (States 50-89)
    // =============================================================================

    50: // FIND_PARKED_VEHICLE
        currentOperation := 'FINDING_VEHICLE';

        IF FindParkedVehicle(VehicleID) THEN
            state := 51;
        ELSE
            Error := TRUE;
            ErrorID := 3001; // Vehicle not found
            state := 90;
        END_IF;

    51: // PREPARE_FOR_RETRIEVAL
        currentOperation := 'PREPARING_RETRIEVAL';

        // Select optimal elevator for retrieval
        selectedElevator := SelectOptimalElevator();

        // Ensure platform is at home
        IF I_Platform_Home THEN
            state := 52;
        ELSE
            MovePlatformToHome();
        END_IF;

    52: // MOVE_TO_RETRIEVAL_LEVEL
        currentOperation := 'MOVING_TO_LEVEL';

        targetLevel := optimalSpace.Level;
        MoveElevatorToLevel(selectedElevator, targetLevel);

        // Check if elevator reached target level
        CASE selectedElevator OF
            1: IF ABS(AI_Elevator1_Position - (targetLevel * 3000)) < 50 THEN
                   state := 53;
               END_IF;
            2: IF ABS(AI_Elevator2_Position - (targetLevel * 3000)) < 50 THEN
                   state := 53;
               END_IF;
            3: IF ABS(AI_Elevator3_Position - (targetLevel * 3000)) < 50 THEN
                   state := 53;
               END_IF;
        END_CASE;

    53: // MOVE_PLATFORM_TO_VEHICLE
        currentOperation := 'MOVING_TO_VEHICLE';

        targetXPosition := optimalSpace.Position * 300.0;
        targetYPosition := 7500.0;

        MovePlatformToPosition(targetXPosition, targetYPosition, 0.0);

        IF ABS(AI_Platform_XPosition - targetXPosition) < 10 AND
           ABS(AI_Platform_YPosition - targetYPosition) < 10 THEN
            state := 54;
        END_IF;

    54: // PICKUP_VEHICLE
        currentOperation := 'PICKING_UP_VEHICLE';

        stepTimer(IN := TRUE, PT := T#30s);

        // Raise platform to pickup vehicle
        Q_Platform_ZDirection := TRUE; // Move up
        AQ_Platform_ZSpeedRef := 200; // Slow speed for safety

        // Check if vehicle picked up (increased weight)
        IF AI_LoadCell_PlatformWeight > 500 THEN
            Platform.VehicleSecured := TRUE;
            state := 55;
            stepTimer(IN := FALSE);
        ELSIF stepTimer.Q THEN
            Error := TRUE;
            ErrorID := 3002; // Vehicle pickup timeout
            state := 90;
            stepTimer(IN := FALSE);
        END_IF;

    55: // MOVE_TO_ELEVATOR_FOR_RETRIEVAL
        currentOperation := 'MOVING_TO_ELEVATOR';

        // Calculate elevator position
        CASE selectedElevator OF
            1: targetXPosition := 1500.0;
            2: targetXPosition := 3000.0;
            3: targetXPosition := 4500.0;
        END_CASE;

        targetYPosition := 2000.0;

        MovePlatformToPosition(targetXPosition, targetYPosition, Platform.ZPosition);

        IF ABS(AI_Platform_XPosition - targetXPosition) < 20 AND
           ABS(AI_Platform_YPosition - targetYPosition) < 20 THEN
            state := 56;
        END_IF;

    56: // LOAD_INTO_ELEVATOR_FOR_RETRIEVAL
        currentOperation := 'LOADING_INTO_ELEVATOR';

        stepTimer(IN := TRUE, PT := T#60s);

        // Move platform into elevator
        Q_Platform_YDirection := TRUE;
        AQ_Platform_YSpeedRef := 500;

        IF ABS(AI_Platform_YPosition - 1000.0) < 10 THEN
            state := 57;
            stepTimer(IN := FALSE);
        ELSIF stepTimer.Q THEN
            Error := TRUE;
            ErrorID := 3003; // Elevator loading timeout
            state := 90;
            stepTimer(IN := FALSE);
        END_IF;

    57: // MOVE_TO_GROUND_LEVEL
        currentOperation := 'MOVING_TO_GROUND';

        MoveElevatorToLevel(selectedElevator, 1); // Ground level

        // Check if elevator reached ground level
        CASE selectedElevator OF
            1: IF ABS(AI_Elevator1_Position) < 50 THEN
                   state := 58;
               END_IF;
            2: IF ABS(AI_Elevator2_Position) < 50 THEN
                   state := 58;
               END_IF;
            3: IF ABS(AI_Elevator3_Position) < 50 THEN
                   state := 58;
               END_IF;
        END_CASE;

    58: // UNLOAD_FROM_ELEVATOR_TO_EXIT
        currentOperation := 'UNLOADING_FOR_EXIT';

        stepTimer(IN := TRUE, PT := T#60s);

        // Move platform out of elevator
        Q_Platform_YDirection := FALSE;
        targetYPosition := 15000.0; // Exit position

        IF ABS(AI_Platform_YPosition - targetYPosition) < 20 THEN
            state := 59;
            stepTimer(IN := FALSE);
        ELSIF stepTimer.Q THEN
            Error := TRUE;
            ErrorID := 3004; // Exit positioning timeout
            state := 90;
            stepTimer(IN := FALSE);
        END_IF;

    59: // DELIVER_VEHICLE
        currentOperation := 'DELIVERING_VEHICLE';

        stepTimer(IN := TRUE, PT := T#30s);

        // Lower platform to deliver vehicle
        Q_Platform_ZDirection := FALSE;
        AQ_Platform_ZSpeedRef := 200;

        // Check if vehicle delivered
        IF AI_LoadCell_PlatformWeight < 100 THEN
            state := 60;
            stepTimer(IN := FALSE);
        ELSIF stepTimer.Q THEN
            Error := TRUE;
            ErrorID := 3005; // Vehicle delivery timeout
            state := 90;
            stepTimer(IN := FALSE);
        END_IF;

    60: // UPDATE_RETRIEVAL_RECORD
        currentOperation := 'UPDATING_RECORDS';

        // Mark space as available
        ParkingSpaces[optimalSpace.Level, optimalSpace.Position].Occupied := FALSE;
        ParkingSpaces[optimalSpace.Level, optimalSpace.Position].VehicleID := '';

        // Update system statistics
        SystemStats.TotalVehiclesRetrieved := SystemStats.TotalVehiclesRetrieved + 1;
        retrievalSequenceTime := operationTimer.ET;

        state := 61; // Return platform home

    61: // RETURN_PLATFORM_HOME_AFTER_RETRIEVAL
        currentOperation := 'RETURNING_HOME';

        MovePlatformToHome();

        IF I_Platform_Home THEN
            state := 70; // Retrieval complete
        END_IF;

    70: // RETRIEVAL_COMPLETE
        currentOperation := 'RETRIEVAL_COMPLETE';
        Done := TRUE;
        Busy := FALSE;
        state := 0;

        // Log successful retrieval
        LogEvent('RETRIEVAL_SUCCESS', VehicleID + ' retrieved from Level ' +
                 INT_TO_STRING(optimalSpace.Level) + ' Position ' +
                 INT_TO_STRING(optimalSpace.Position));

    // =============================================================================
    // ERROR HANDLING (States 90-99)
    // =============================================================================

    90: // ERROR_STATE
        currentOperation := 'ERROR_HANDLING';
        Error := TRUE;
        Busy := FALSE;

        // Log error
        LogError(ErrorID, 'Parking Controller Error: ' + INT_TO_STRING(ErrorID));

        // Attempt recovery if retries available
        IF retryCount < maxRetries THEN
            retryCount := retryCount + 1;
            stepTimer(IN := TRUE, PT := T#5s);
            IF stepTimer.Q THEN
                state := 10; // Retry from beginning
                stepTimer(IN := FALSE);
            END_IF;
        ELSE
            state := 0; // Give up and return to idle
            retryCount := 0;
        END_IF;

END_CASE;

// ============================================================================
// HELPER FUNCTIONS
// ============================================================================

// Function to find optimal parking space
FUNCTION FindOptimalParkingSpace : BOOL
VAR
    level, position : INT;
    found : BOOL := FALSE;
    bestLevel, bestPosition : INT;
    minDistance : REAL := 999999.0;
    distance : REAL;
END_VAR

// Search for available space starting from lowest levels
FOR level := 1 TO MAX_PARKING_LEVELS DO
    FOR position := 1 TO SPACES_PER_LEVEL DO
        IF NOT ParkingSpaces[level, position].Occupied AND
           NOT ParkingSpaces[level, position].MaintenanceRequired THEN

            // Calculate distance/efficiency score
            distance := level * 100.0 + ABS(position - 10) * 10.0;

            IF distance < minDistance THEN
                minDistance := distance;
                bestLevel := level;
                bestPosition := position;
                found := TRUE;
            END_IF;
        END_IF;
    END_FOR;
END_FOR;

IF found THEN
    optimalSpace.Level := bestLevel;
    optimalSpace.Position := bestPosition;
    spaceAvailable := TRUE;
ELSE
    spaceAvailable := FALSE;
END_IF;

FindOptimalParkingSpace := found;
END_FUNCTION;

// Function to select optimal elevator
FUNCTION SelectOptimalElevator : INT
VAR
    selectedElev : INT := 0;
    elev1Distance, elev2Distance, elev3Distance : REAL;
    targetPosition : REAL;
END_VAR

targetPosition := targetLevel * 3000.0;

// Calculate distance for each elevator
elev1Distance := ABS(AI_Elevator1_Position - targetPosition);
elev2Distance := ABS(AI_Elevator2_Position - targetPosition);
elev3Distance := ABS(AI_Elevator3_Position - targetPosition);

// Select closest available elevator
IF Elevator1.Available AND (elev1Distance <= elev2Distance) AND (elev1Distance <= elev3Distance) THEN
    selectedElev := 1;
ELSIF Elevator2.Available AND (elev2Distance <= elev3Distance) THEN
    selectedElev := 2;
ELSIF Elevator3.Available THEN
    selectedElev := 3;
END_IF;

SelectOptimalElevator := selectedElev;
END_FUNCTION;

// Calculate estimated operation time
EstimatedTime := T#90s; // Base time
IF vehicleDimensions.VehicleType = SUV THEN
    EstimatedTime := EstimatedTime + T#30s; // Extra time for larger vehicles
END_IF;
IF targetLevel > 10 THEN
    EstimatedTime := EstimatedTime + T#20s; // Extra time for higher levels
END_IF;

END_FUNCTION_BLOCK

(* ---- payment_controller.st ---- *)
FUNCTION_BLOCK PaymentController
VAR_INPUT
    ProcessPayment : BOOL;              // Start payment processing
    CustomerID : STRING[50];            // Customer identification
    RequestedDuration : TIME;           // Requested parking duration
    VehicleType : VehicleSize;          // Vehicle size category
    CancelPayment : BOOL;               // Cancel current transaction
END_VAR

VAR_OUTPUT
    PaymentComplete : BOOL;             // Payment successfully processed
    PaymentAmount : REAL;               // Total amount charged
    PaymentMethod : PaymentMethod;      // Method used for payment
    TransactionID : DINT;               // Unique transaction identifier
    ReceiptPrinted : BOOL;              // Receipt printing status
    Error : BOOL;                       // Payment error occurred
    ErrorCode : INT;                    // Payment error code
    TimeRemaining : TIME;               // Time remaining for payment
END_VAR

VAR
    // Payment state machine
    paymentState : INT := 0;
    stateTimer : TON;
    paymentTimer : TON;

    // Payment processing
    calculatedAmount : REAL;
    discountApplied : REAL := 0.0;
    taxAmount : REAL := 0.0;
    totalAmount : REAL;

    // Payment methods status
    cashAmount : REAL := 0.0;
    cardTransactionActive : BOOL := FALSE;
    rfidBalance : REAL := 0.0;
    mobilePaymentPending : BOOL := FALSE;

    // Customer interface
    displayMessage : STRING[100];
    keypadInput : STRING[20];
    selectedMethod : PaymentMethod := NONE;

    // Receipt and ticket data
    ticketData : TicketInfo;
    receiptData : ReceiptInfo;

    // Retry and timeout handling
    retryCount : INT := 0;
    maxRetries : INT := 3;
    paymentTimeout : TIME := T#120s;

    // Security and validation
    cardValidated : BOOL := FALSE;
    pinVerified : BOOL := FALSE;
    securityCode : STRING[10];

END_VAR

// Payment data structures
TYPE TicketInfo :
STRUCT
    TicketNumber : STRING[20];
    IssueTime : DATE_AND_TIME;
    ExpiryTime : DATE_AND_TIME;
    CustomerID : STRING[50];
    VehicleID : STRING[20];
    ParkingLevel : INT;
    ParkingPosition : INT;
    Amount : REAL;
    PaymentMethod : STRING[20];
    QRCode : STRING[100];
END_STRUCT;
END_TYPE;

TYPE ReceiptInfo :
STRUCT
    ReceiptNumber : STRING[20];
    TransactionTime : DATE_AND_TIME;
    MerchantID : STRING[20];
    Amount : REAL;
    Tax : REAL;
    Total : REAL;
    PaymentMethod : STRING[20];
    AuthorizationCode : STRING[20];
END_STRUCT;
END_TYPE;

// Initialize payment processing
IF ProcessPayment AND paymentState = 0 THEN
    paymentState := 10; // Start payment sequence
    paymentTimer(IN := TRUE, PT := paymentTimeout);
    TransactionCounter := TransactionCounter + 1;
    TransactionID := TransactionCounter;
    Error := FALSE;
    ErrorCode := 0;
    PaymentComplete := FALSE;
END_IF;

// Cancel payment if requested
IF CancelPayment THEN
    paymentState := 90; // Cancel state
    PaymentComplete := FALSE;
    Error := TRUE;
    ErrorCode := 4999; // Payment cancelled
END_IF;

// Payment timeout handling
paymentTimer(IN := paymentState > 0 AND paymentState < 80, PT := paymentTimeout);
TimeRemaining := paymentTimeout - paymentTimer.ET;

IF paymentTimer.Q AND paymentState > 0 AND paymentState < 80 THEN
    paymentState := 91; // Timeout state
    Error := TRUE;
    ErrorCode := 4001; // Payment timeout
END_IF;

// Main payment state machine
CASE paymentState OF

    0: // IDLE
        PaymentComplete := FALSE;
        Error := FALSE;
        displayMessage := 'System Ready';

    // =============================================================================
    // PAYMENT INITIALIZATION (States 10-19)
    // =============================================================================

    10: // CALCULATE_AMOUNT
        displayMessage := 'Calculating parking fee...';

        // Base calculation on duration and vehicle type
        IF RequestedDuration <= T#1h THEN
            calculatedAmount := HourlyRate;
        ELSIF RequestedDuration <= T#24h THEN
            calculatedAmount := REAL_TO_TIME(RequestedDuration) / 3600000.0 * HourlyRate;
            IF calculatedAmount > DailyRate THEN
                calculatedAmount := DailyRate; // Daily rate cap
            END_IF;
        ELSE
            calculatedAmount := DailyRate * (REAL_TO_TIME(RequestedDuration) / 86400000.0);
            IF calculatedAmount > MonthlyRate THEN
                calculatedAmount := MonthlyRate; // Monthly rate cap
            END_IF;
        END_IF;

        // Vehicle type surcharge
        CASE VehicleType OF
            COMPACT: calculatedAmount := calculatedAmount * 0.9; // 10% discount
            STANDARD: ; // No change
            SUV: calculatedAmount := calculatedAmount * 1.2; // 20% surcharge
            MOTORCYCLE: calculatedAmount := calculatedAmount * 0.5; // 50% discount
        END_CASE;

        // Apply any customer discounts
        IF CheckCustomerDiscounts(CustomerID) THEN
            discountApplied := calculatedAmount * 0.1; // 10% member discount
            calculatedAmount := calculatedAmount - discountApplied;
        END_IF;

        // Calculate tax
        taxAmount := calculatedAmount * 0.08; // 8% tax
        totalAmount := calculatedAmount + taxAmount;
        PaymentAmount := totalAmount;

        paymentState := 11;

    11: // DISPLAY_AMOUNT_AND_OPTIONS
        displayMessage := 'Amount: $' + REAL_TO_STRING(totalAmount, 2) +
                         ' - Select payment method';

        // Wait for payment method selection
        stateTimer(IN := TRUE, PT := T#30s);

        IF I_CashInserted THEN
            selectedMethod := CASH;
            paymentState := 20; // Cash payment
            stateTimer(IN := FALSE);
        ELSIF I_CardInserted THEN
            selectedMethod := CREDIT_CARD;
            paymentState := 30; // Card payment
            stateTimer(IN := FALSE);
        ELSIF I_RFIDCardPresent THEN
            selectedMethod := RFID_CARD;
            paymentState := 40; // RFID payment
            stateTimer(IN := FALSE);
        ELSIF I_QRCodeScanned THEN
            selectedMethod := MOBILE_APP;
            paymentState := 50; // Mobile payment
            stateTimer(IN := FALSE);
        ELSIF stateTimer.Q THEN
            paymentState := 91; // Selection timeout
            ErrorCode := 4002;
            stateTimer(IN := FALSE);
        END_IF;

    // =============================================================================
    // CASH PAYMENT (States 20-29)
    // =============================================================================

    20: // PROCESS_CASH_PAYMENT
        displayMessage := 'Insert cash: $' + REAL_TO_STRING(totalAmount, 2);
        PaymentMethod := CASH;

        stateTimer(IN := TRUE, PT := T#60s);

        // Simulate cash counting (in real system, would interface with bill acceptor)
        cashAmount := GetCashAmount();

        IF cashAmount >= totalAmount THEN
            paymentState := 21; // Sufficient cash received
            stateTimer(IN := FALSE);
        ELSIF stateTimer.Q THEN
            paymentState := 92; // Cash timeout
            ErrorCode := 4003;
            stateTimer(IN := FALSE);
        END_IF;

    21: // CALCULATE_CHANGE
        displayMessage := 'Processing cash payment...';

        IF cashAmount > totalAmount THEN
            // Dispense change
            Q_CashDispenser_Enable := TRUE;
            stateTimer(IN := TRUE, PT := T#10s);

            IF stateTimer.Q THEN
                displayMessage := 'Change dispensed: $' +
                                REAL_TO_STRING(cashAmount - totalAmount, 2);
                paymentState := 70; // Payment complete
                stateTimer(IN := FALSE);
            END_IF;
        ELSE
            paymentState := 70; // Exact change
        END_IF;

    // =============================================================================
    // CREDIT/DEBIT CARD PAYMENT (States 30-39)
    // =============================================================================

    30: // PROCESS_CARD_PAYMENT
        displayMessage := 'Processing card...';
        PaymentMethod := CREDIT_CARD;

        Q_CardReader_Enable := TRUE;
        cardTransactionActive := TRUE;

        stateTimer(IN := TRUE, PT := T#30s);

        // Simulate card validation
        IF ValidateCard() THEN
            paymentState := 31;
            stateTimer(IN := FALSE);
        ELSIF stateTimer.Q THEN
            paymentState := 93; // Card timeout
            ErrorCode := 4004;
            stateTimer(IN := FALSE);
        END_IF;

    31: // REQUEST_PIN
        displayMessage := 'Enter PIN';

        stateTimer(IN := TRUE, PT := T#60s);

        // Get PIN from keypad (simulated)
        IF GetPINInput() THEN
            IF VerifyPIN() THEN
                paymentState := 32;
                stateTimer(IN := FALSE);
            ELSE
                retryCount := retryCount + 1;
                IF retryCount >= maxRetries THEN
                    paymentState := 94; // PIN failed
                    ErrorCode := 4005;
                ELSE
                    displayMessage := 'Incorrect PIN - Try again';
                END_IF;
            END_IF;
        ELSIF stateTimer.Q THEN
            paymentState := 93; // PIN timeout
            ErrorCode := 4006;
            stateTimer(IN := FALSE);
        END_IF;

    32: // AUTHORIZE_TRANSACTION
        displayMessage := 'Authorizing transaction...';

        stateTimer(IN := TRUE, PT := T#20s);

        // Simulate bank authorization
        IF AuthorizeCardTransaction(totalAmount) THEN
            receiptData.AuthorizationCode := GenerateAuthCode();
            paymentState := 70; // Payment approved
            stateTimer(IN := FALSE);
        ELSIF stateTimer.Q THEN
            paymentState := 95; // Authorization failed
            ErrorCode := 4007;
            stateTimer(IN := FALSE);
        END_IF;

    // =============================================================================
    // RFID CARD PAYMENT (States 40-49)
    // =============================================================================

    40: // PROCESS_RFID_PAYMENT
        displayMessage := 'Reading RFID card...';
        PaymentMethod := RFID_CARD;

        stateTimer(IN := TRUE, PT := T#10s);

        // Read RFID card balance
        rfidBalance := GetRFIDBalance(CustomerID);

        IF rfidBalance >= totalAmount THEN
            paymentState := 41;
            stateTimer(IN := FALSE);
        ELSIF stateTimer.Q THEN
            paymentState := 96; // Insufficient RFID balance
            ErrorCode := 4008;
            stateTimer(IN := FALSE);
        END_IF;

    41: // DEDUCT_RFID_BALANCE
        displayMessage := 'Deducting from RFID card...';

        stateTimer(IN := TRUE, PT := T#5s);

        IF DeductRFIDBalance(CustomerID, totalAmount) THEN
            paymentState := 70; // Payment complete
            stateTimer(IN := FALSE);
        ELSE
            paymentState := 97; // RFID deduction failed
            ErrorCode := 4009;
            stateTimer(IN := FALSE);
        END_IF;

    // =============================================================================
    // MOBILE/QR CODE PAYMENT (States 50-59)
    // =============================================================================

    50: // PROCESS_MOBILE_PAYMENT
        displayMessage := 'Processing mobile payment...';
        PaymentMethod := MOBILE_APP;

        mobilePaymentPending := TRUE;
        stateTimer(IN := TRUE, PT := T#45s);

        // Wait for mobile payment confirmation
        IF CheckMobilePaymentStatus() THEN
            paymentState := 70; // Payment confirmed
            stateTimer(IN := FALSE);
        ELSIF stateTimer.Q THEN
            paymentState := 98; // Mobile payment timeout
            ErrorCode := 4010;
            stateTimer(IN := FALSE);
        END_IF;

    // =============================================================================
    // PAYMENT COMPLETION (States 70-79)
    // =============================================================================

    70: // PAYMENT_SUCCESSFUL
        displayMessage := 'Payment approved - Printing ticket...';

        // Generate parking ticket
        GenerateTicket();

        // Print ticket
        IF I_TicketPrinter_Ready AND I_TicketPrinter_PaperOK THEN
            Q_TicketPrinter_Print := TRUE;
            paymentState := 71;
        ELSE
            paymentState := 99; // Printer error
            ErrorCode := 4011;
        END_IF;

    71: // PRINT_RECEIPT
        displayMessage := 'Printing receipt...';

        // Generate receipt
        GenerateReceipt();

        stateTimer(IN := TRUE, PT := T#10s);

        IF I_ReceiptPrinter_Ready THEN
            Q_ReceiptPrinter_Print := TRUE;
            ReceiptPrinted := TRUE;
            paymentState := 72;
            stateTimer(IN := FALSE);
        ELSIF stateTimer.Q THEN
            // Continue without receipt if printer fails
            ReceiptPrinted := FALSE;
            paymentState := 72;
            stateTimer(IN := FALSE);
        END_IF;

    72: // UPDATE_TRANSACTION_RECORD
        displayMessage := 'Transaction complete';

        // Update current transaction
        CurrentTransaction.TransactionID := TransactionID;
        CurrentTransaction.Timestamp := GetSystemTime();
        CurrentTransaction.CustomerID := CustomerID;
        CurrentTransaction.PaymentMethod := selectedMethod;
        CurrentTransaction.Amount := totalAmount;
        CurrentTransaction.ParkingDuration := RequestedDuration;
        CurrentTransaction.Status := 'PAID';

        // Update system statistics
        SystemStats.TotalRevenue := SystemStats.TotalRevenue + totalAmount;

        PaymentComplete := TRUE;
        paymentState := 0; // Return to idle

        // Log successful payment
        LogEvent('PAYMENT_SUCCESS', 'Customer: ' + CustomerID +
                 ', Amount: $' + REAL_TO_STRING(totalAmount, 2) +
                 ', Method: ' + PaymentMethodToString(selectedMethod));

    // =============================================================================
    // ERROR STATES (States 90-99)
    // =============================================================================

    90: // PAYMENT_CANCELLED
        displayMessage := 'Payment cancelled';
        Error := TRUE;
        PaymentComplete := FALSE;

        // Refund any partial payments
        IF selectedMethod = CASH AND cashAmount > 0 THEN
            Q_CashDispenser_Enable := TRUE; // Return cash
        END_IF;

        stateTimer(IN := TRUE, PT := T#5s);
        IF stateTimer.Q THEN
            paymentState := 0; // Return to idle
            stateTimer(IN := FALSE);
        END_IF;

    91: // PAYMENT_TIMEOUT
        displayMessage := 'Payment timeout - Please try again';
        Error := TRUE;
        PaymentComplete := FALSE;

        stateTimer(IN := TRUE, PT := T#10s);
        IF stateTimer.Q THEN
            paymentState := 0;
            stateTimer(IN := FALSE);
        END_IF;

    92: // CASH_TIMEOUT
        displayMessage := 'Cash insertion timeout';
        Error := TRUE;

        // Return any inserted cash
        IF cashAmount > 0 THEN
            Q_CashDispenser_Enable := TRUE;
        END_IF;

        stateTimer(IN := TRUE, PT := T#10s);
        IF stateTimer.Q THEN
            paymentState := 0;
            stateTimer(IN := FALSE);
        END_IF;

    93: // CARD_ERROR
        displayMessage := 'Card error - Please try again';
        Error := TRUE;
        cardTransactionActive := FALSE;
        Q_CardReader_Enable := FALSE;

        stateTimer(IN := TRUE, PT := T#10s);
        IF stateTimer.Q THEN
            paymentState := 0;
            stateTimer(IN := FALSE);
        END_IF;

    94: // PIN_ERROR
        displayMessage := 'PIN verification failed';
        Error := TRUE;
        cardTransactionActive := FALSE;

        stateTimer(IN := TRUE, PT := T#10s);
        IF stateTimer.Q THEN
            paymentState := 0;
            retryCount := 0;
            stateTimer(IN := FALSE);
        END_IF;

    95: // AUTHORIZATION_FAILED
        displayMessage := 'Transaction declined';
        Error := TRUE;
        cardTransactionActive := FALSE;

        stateTimer(IN := TRUE, PT := T#10s);
        IF stateTimer.Q THEN
            paymentState := 0;
            stateTimer(IN := FALSE);
        END_IF;

    96: // INSUFFICIENT_RFID_BALANCE
        displayMessage := 'Insufficient card balance: $' + REAL_TO_STRING(rfidBalance, 2);
        Error := TRUE;

        stateTimer(IN := TRUE, PT := T#10s);
        IF stateTimer.Q THEN
            paymentState := 0;
            stateTimer(IN := FALSE);
        END_IF;

    97: // RFID_ERROR
        displayMessage := 'RFID card error';
        Error := TRUE;

        stateTimer(IN := TRUE, PT := T#10s);
        IF stateTimer.Q THEN
            paymentState := 0;
            stateTimer(IN := FALSE);
        END_IF;

    98: // MOBILE_PAYMENT_ERROR
        displayMessage := 'Mobile payment failed';
        Error := TRUE;
        mobilePaymentPending := FALSE;

        stateTimer(IN := TRUE, PT := T#10s);
        IF stateTimer.Q THEN
            paymentState := 0;
            stateTimer(IN := FALSE);
        END_IF;

    99: // PRINTER_ERROR
        displayMessage := 'Printer error - Payment successful';
        Error := FALSE; // Payment was successful, just printer issue
        PaymentComplete := TRUE;

        stateTimer(IN := TRUE, PT := T#5s);
        IF stateTimer.Q THEN
            paymentState := 0;
            stateTimer(IN := FALSE);
        END_IF;

END_CASE;

// ============================================================================
// HELPER FUNCTIONS
// ============================================================================

FUNCTION GenerateTicket : BOOL
ticketData.TicketNumber := 'PKT' + INT_TO_STRING(TransactionID);
ticketData.IssueTime := GetSystemTime();
ticketData.ExpiryTime := ticketData.IssueTime + RequestedDuration;
ticketData.CustomerID := CustomerID;
ticketData.Amount := totalAmount;
ticketData.PaymentMethod := PaymentMethodToString(selectedMethod);
ticketData.QRCode := GenerateQRCode(ticketData.TicketNumber);
GenerateTicket := TRUE;
END_FUNCTION;

FUNCTION GenerateReceipt : BOOL
receiptData.ReceiptNumber := 'RCP' + INT_TO_STRING(TransactionID);
receiptData.TransactionTime := GetSystemTime();
receiptData.MerchantID := 'PARK001';
receiptData.Amount := calculatedAmount;
receiptData.Tax := taxAmount;
receiptData.Total := totalAmount;
receiptData.PaymentMethod := PaymentMethodToString(selectedMethod);
GenerateReceipt := TRUE;
END_FUNCTION;

FUNCTION PaymentMethodToString : STRING
CASE selectedMethod OF
    CASH: PaymentMethodToString := 'CASH';
    CREDIT_CARD: PaymentMethodToString := 'CREDIT CARD';
    RFID_CARD: PaymentMethodToString := 'RFID CARD';
    MOBILE_APP: PaymentMethodToString := 'MOBILE APP';
    QR_CODE: PaymentMethodToString := 'QR CODE';
    ELSE: PaymentMethodToString := 'UNKNOWN';
END_CASE;
END_FUNCTION;

// Clean up on completion
IF paymentState = 0 THEN
    Q_TicketPrinter_Print := FALSE;
    Q_ReceiptPrinter_Print := FALSE;
    Q_CashDispenser_Enable := FALSE;
    Q_CardReader_Enable := FALSE;
    cashAmount := 0.0;
    cardTransactionActive := FALSE;
    mobilePaymentPending := FALSE;
    selectedMethod := NONE;
END_IF;

END_FUNCTION_BLOCK

(* ---- safety_controller.st ---- *)
(*
===============================================================================
SAFETY CONTROLLER
===============================================================================
Purpose: Emergency procedures, safety interlocks, and fail-safe operations
Author: Industrial Automation System
Date: June 8, 2025
Version: 1.0

Safety Requirements:
- Emergency stop activation within 1 second
- Fire suppression system activation
- Elevator emergency brake engagement
- Personnel safety zone monitoring
- Automatic ventilation control
- Emergency lighting activation
- Communication with emergency services
===============================================================================
*)

FUNCTION_BLOCK SafetyController
VAR_INPUT
    Enable : BOOL;                      // Enable safety monitoring
    Reset : BOOL;                       // Reset safety alarms
    TestMode : BOOL;                    // Safety system test mode
END_VAR

VAR_OUTPUT
    SafetyOK : BOOL;                    // Overall safety status
    EmergencyActive : BOOL;             // Emergency condition active
    EvacuationRequired : BOOL;          // Evacuation alarm active
    MaintenanceRequired : BOOL;         // Safety maintenance needed
    SafetyAlarm : BOOL;                 // Safety alarm output
END_VAR

VAR
    // Emergency Stop Processing
    EmergencyStopChain : BOOL;          // Emergency stop chain status
    EmergencyStopTimer : TON;           // Emergency stop response timer
    EmergencyResetTimer : TON;          // Emergency reset delay timer

    // Fire Safety System
    FireDetected : BOOL;                // Fire detection status
    FireSuppressionActive : BOOL;       // Fire suppression system active
    EvacuationTimer : TON;              // Evacuation countdown timer
    FireZoneStatus : ARRAY[1..15] OF BOOL; // Fire status per level

    // Personnel Safety
    PersonnelInZone : ARRAY[1..10] OF BOOL; // Personnel detection zones
    SafetyZoneViolation : BOOL;         // Safety zone violation detected
    AccessControlActive : BOOL;         // Access control system status

    // Equipment Safety Interlocks
    ElevatorSafetyOK : ARRAY[1..3] OF BOOL;  // Elevator safety status
    PlatformSafetyOK : ARRAY[1..20] OF BOOL; // Platform safety status
    MotorSafetyOK : BOOL;               // Motor safety interlocks
    HydraulicSafetyOK : BOOL;           // Hydraulic system safety

    // Environmental Safety
    VentilationStatus : BOOL;           // Ventilation system status
    CO_LevelOK : BOOL;                  // Carbon monoxide levels OK
    TemperatureOK : BOOL;               // Temperature within safe limits
    HumidityOK : BOOL;                  // Humidity within safe limits

    // Communication Safety
    PLCHeartbeat : BOOL;                // PLC communication heartbeat
    HMIHeartbeat : BOOL;                // HMI communication heartbeat
    NetworkStatus : BOOL;               // Network communication status

    // Safety State Machine
    SafetyState : INT;                  // Current safety state
    PreviousState : INT;                // Previous safety state
    StateTimer : TON;                   // State transition timer

    // Diagnostic Variables
    SafetyTestResults : ARRAY[1..20] OF BOOL; // Safety test results
    LastTestTime : DATE_AND_TIME;       // Last safety test timestamp
    TestInProgress : BOOL;              // Safety test in progress

    // Counters and Statistics
    EmergencyStopCount : DINT;          // Emergency stop activation count
    FireAlarmCount : DINT;              // Fire alarm activation count
    SafetyViolationCount : DINT;        // Safety violation count
    SystemUptimeHours : DINT;           // System uptime in hours
END_VAR

// Safety State Definitions
VAR CONSTANT
    SAFETY_NORMAL : INT := 0;           // Normal operation
    SAFETY_WARNING : INT := 1;          // Warning condition
    SAFETY_ALARM : INT := 2;            // Alarm condition
    SAFETY_EMERGENCY : INT := 3;        // Emergency condition
    SAFETY_EVACUATION : INT := 4;       // Evacuation required
    SAFETY_LOCKDOWN : INT := 5;         // System lockdown
    SAFETY_TEST : INT := 6;             // Safety test mode
    SAFETY_MAINTENANCE : INT := 7;      // Maintenance mode
END_VAR

// Main Safety Controller Logic
IF NOT Enable THEN
    SafetyOK := FALSE;
    SafetyState := SAFETY_LOCKDOWN;
    RETURN;
END_IF

// Emergency Stop Chain Monitoring
EmergencyStopChain := Emergency_Stop_Main AND
                      Emergency_Stop_Level1 AND
                      Emergency_Stop_Level2 AND
                      Emergency_Stop_Maintenance AND
                      Emergency_Stop_HMI;

// Emergency Stop Processing
IF NOT EmergencyStopChain THEN
    EmergencyActive := TRUE;
    SafetyState := SAFETY_EMERGENCY;
    EmergencyStopCount := EmergencyStopCount + 1;

    // Activate emergency procedures
    Emergency_Elevator_Stop := TRUE;
    Emergency_Platform_Stop := TRUE;
    Emergency_Motor_Stop := TRUE;
    Emergency_Lighting := TRUE;
    Emergency_Ventilation := TRUE;

    // Start emergency response timer
    EmergencyStopTimer(IN := TRUE, PT := T#1S);
END_IF

// Fire Detection and Suppression
FireDetected := Fire_Detector_Level1 OR Fire_Detector_Level2 OR
                Fire_Detector_Basement OR Smoke_Detector_Main OR
                Heat_Detector_Electrical;

IF FireDetected THEN
    SafetyState := SAFETY_EVACUATION;
    EvacuationRequired := TRUE;
    FireAlarmCount := FireAlarmCount + 1;

    // Activate fire suppression sequence
    Fire_Suppression_Activate := TRUE;
    Emergency_Ventilation := TRUE;
    Evacuation_Alarm := TRUE;
    Emergency_Lighting := TRUE;

    // Evacuate all vehicles from affected zones
    IF Fire_Detector_Level1 THEN
        Evacuate_Level_1 := TRUE;
    END_IF
    IF Fire_Detector_Level2 THEN
        Evacuate_Level_2 := TRUE;
    END_IF

    // Start evacuation timer (10 minutes)
    EvacuationTimer(IN := TRUE, PT := T#10M);
END_IF

// Personnel Safety Zone Monitoring
SafetyZoneViolation := FALSE;
FOR i := 1 TO 10 DO
    IF PersonnelInZone[i] AND Equipment_Operating THEN
        SafetyZoneViolation := TRUE;
        SafetyViolationCount := SafetyViolationCount + 1;
    END_IF
END_FOR

// Equipment Safety Interlocks
FOR i := 1 TO 3 DO
    ElevatorSafetyOK[i] := Elevator_Door_Closed[i] AND
                           Elevator_Position_Valid[i] AND
                           Elevator_Speed_Safe[i] AND
                           Elevator_Load_Safe[i];
END_FOR

FOR i := 1 TO 20 DO
    PlatformSafetyOK[i] := Platform_Position_Valid[i] AND
                           Platform_Load_Safe[i] AND
                           Platform_Clear[i];
END_FOR

// Motor Safety Interlocks
MotorSafetyOK := Motor_Temperature_OK AND
                 Motor_Current_OK AND
                 Motor_Vibration_OK AND
                 Motor_Overload_OK;

// Hydraulic System Safety
HydraulicSafetyOK := Hydraulic_Pressure_OK AND
                     Hydraulic_Temperature_OK AND
                     Hydraulic_Level_OK AND
                     Hydraulic_Filter_OK;

// Environmental Safety Monitoring
VentilationStatus := Ventilation_Fan_1_OK AND
                     Ventilation_Fan_2_OK AND
                     Air_Quality_OK;

CO_LevelOK := CO_Level < 35;  // ppm limit
TemperatureOK := (Ambient_Temperature > 5) AND (Ambient_Temperature < 40);
HumidityOK := (Relative_Humidity > 20) AND (Relative_Humidity < 80);

// Communication Safety Heartbeat
PLCHeartbeat := PLC_Status_OK;
HMIHeartbeat := HMI_Status_OK;
NetworkStatus := Network_Status_OK;

// Safety State Machine
CASE SafetyState OF
    SAFETY_NORMAL:
        IF TestMode THEN
            SafetyState := SAFETY_TEST;
        ELSIF FireDetected THEN
            SafetyState := SAFETY_EVACUATION;
        ELSIF NOT EmergencyStopChain THEN
            SafetyState := SAFETY_EMERGENCY;
        ELSIF SafetyZoneViolation THEN
            SafetyState := SAFETY_WARNING;
        END_IF

    SAFETY_WARNING:
        SafetyAlarm := TRUE;
        IF NOT SafetyZoneViolation THEN
            SafetyState := SAFETY_NORMAL;
        ELSIF EmergencyStopChain = FALSE THEN
            SafetyState := SAFETY_EMERGENCY;
        END_IF

    SAFETY_ALARM:
        SafetyAlarm := TRUE;
        EmergencyActive := TRUE;
        IF Reset AND (NOT FireDetected) AND EmergencyStopChain THEN
            EmergencyResetTimer(IN := TRUE, PT := T#5S);
            IF EmergencyResetTimer.Q THEN
                SafetyState := SAFETY_NORMAL;
                EmergencyResetTimer(IN := FALSE);
            END_IF
        END_IF

    SAFETY_EMERGENCY:
        EmergencyActive := TRUE;
        SafetyAlarm := TRUE;

        // All equipment emergency stop
        Emergency_All_Stop := TRUE;

        IF Reset AND EmergencyStopChain AND (NOT FireDetected) THEN
            EmergencyResetTimer(IN := TRUE, PT := T#10S);
            IF EmergencyResetTimer.Q THEN
                SafetyState := SAFETY_NORMAL;
                EmergencyActive := FALSE;
                Emergency_All_Stop := FALSE;
                EmergencyResetTimer(IN := FALSE);
            END_IF
        END_IF

    SAFETY_EVACUATION:
        EvacuationRequired := TRUE;
        EmergencyActive := TRUE;
        SafetyAlarm := TRUE;

        // Complete system shutdown
        Emergency_All_Stop := TRUE;
        Evacuation_Alarm := TRUE;
        Emergency_Lighting := TRUE;

        // Automatic fire department notification
        Fire_Department_Alert := TRUE;

        EvacuationTimer(IN := TRUE, PT := T#30M);
        IF EvacuationTimer.Q AND Reset THEN
            SafetyState := SAFETY_MAINTENANCE;
            EvacuationTimer(IN := FALSE);
        END_IF

    SAFETY_LOCKDOWN:
        EmergencyActive := TRUE;
        SafetyAlarm := TRUE;
        Emergency_All_Stop := TRUE;

        IF Enable AND Reset THEN
            SafetyState := SAFETY_NORMAL;
            EmergencyActive := FALSE;
            Emergency_All_Stop := FALSE;
        END_IF

    SAFETY_TEST:
        TestInProgress := TRUE;

        // Perform safety system tests
        SafetyTestResults[1] := Test_Emergency_Stops();
        SafetyTestResults[2] := Test_Fire_Detection();
        SafetyTestResults[3] := Test_Ventilation();
        SafetyTestResults[4] := Test_Emergency_Lighting();
        SafetyTestResults[5] := Test_Communication();

        StateTimer(IN := TRUE, PT := T#60S);
        IF StateTimer.Q THEN
            TestInProgress := FALSE;
            LastTestTime := NOW();
            SafetyState := SAFETY_NORMAL;
            StateTimer(IN := FALSE);
        END_IF

    SAFETY_MAINTENANCE:
        MaintenanceRequired := TRUE;
        Emergency_All_Stop := TRUE;

        IF Reset AND Maintenance_Complete THEN
            SafetyState := SAFETY_NORMAL;
            MaintenanceRequired := FALSE;
            Emergency_All_Stop := FALSE;
        END_IF
END_CASE

// Overall Safety Status
SafetyOK := (SafetyState = SAFETY_NORMAL) AND
            EmergencyStopChain AND
            (NOT FireDetected) AND
            (NOT SafetyZoneViolation) AND
            MotorSafetyOK AND
            HydraulicSafetyOK AND
            VentilationStatus AND
            CO_LevelOK AND
            TemperatureOK AND
            PLCHeartbeat AND
            HMIHeartbeat;

// Safety Output Assignments
Safety_System_OK := SafetyOK;
Emergency_Stop_Output := EmergencyActive;
Fire_Alarm_Output := FireDetected;
Evacuation_Signal := EvacuationRequired;
Maintenance_Signal := MaintenanceRequired;

END_FUNCTION_BLOCK

(*
===============================================================================
SAFETY SYSTEM TEST FUNCTIONS
===============================================================================
*)

FUNCTION Test_Emergency_Stops : BOOL
VAR
    TestResult : BOOL := TRUE;
END_VAR

// Test all emergency stop circuits
TestResult := TestResult AND Emergency_Stop_Main;
TestResult := TestResult AND Emergency_Stop_Level1;
TestResult := TestResult AND Emergency_Stop_Level2;
TestResult := TestResult AND Emergency_Stop_Maintenance;
TestResult := TestResult AND Emergency_Stop_HMI;

Test_Emergency_Stops := TestResult;
END_FUNCTION

FUNCTION Test_Fire_Detection : BOOL
VAR
    TestResult : BOOL := TRUE;
END_VAR

// Test fire detection systems
TestResult := TestResult AND Fire_Detector_Level1_OK;
TestResult := TestResult AND Fire_Detector_Level2_OK;
TestResult := TestResult AND Smoke_Detector_Main_OK;
TestResult := TestResult AND Heat_Detector_Electrical_OK;

Test_Fire_Detection := TestResult;
END_FUNCTION

FUNCTION Test_Ventilation : BOOL
VAR
    TestResult : BOOL := TRUE;
END_VAR

// Test ventilation systems
TestResult := TestResult AND Ventilation_Fan_1_OK;
TestResult := TestResult AND Ventilation_Fan_2_OK;
TestResult := TestResult AND Emergency_Ventilation_OK;

Test_Ventilation := TestResult;
END_FUNCTION

FUNCTION Test_Emergency_Lighting : BOOL
VAR
    TestResult : BOOL := TRUE;
END_VAR

// Test emergency lighting systems
TestResult := TestResult AND Emergency_Light_1_OK;
TestResult := TestResult AND Emergency_Light_2_OK;
TestResult := TestResult AND Exit_Light_1_OK;
TestResult := TestResult AND Exit_Light_2_OK;

Test_Emergency_Lighting := TestResult;
END_FUNCTION

FUNCTION Test_Communication : BOOL
VAR
    TestResult : BOOL := TRUE;
END_VAR

// Test communication systems
TestResult := TestResult AND PLC_Status_OK;
TestResult := TestResult AND HMI_Status_OK;
TestResult := TestResult AND Network_Status_OK;
TestResult := TestResult AND Fire_Department_Comm_OK;

Test_Communication := TestResult;
END_FUNCTION
